% RSLogix 500 project ML02B JOB 10 NL.RSS, saved by version 10.00.00.00 %
PROJECT "UNTITLED"    % processor: Bul.1763 MicroLogix 1100 Series B %

PROGRAM FILES
  LAD 2   5 rungs

DATA FILES
  O0 OUTPUT  4 elements
  I1 INPUT  6 elements
  S2 STATUS  66 elements
  B3 BINARY  1 elements
  T4 TIMER  1 elements
  C5 COUNTER  1 elements
  R6 CONTROL  1 elements
  N7 INTEGER  1 elements
  F8 FLOAT  1 elements

LADDER 2
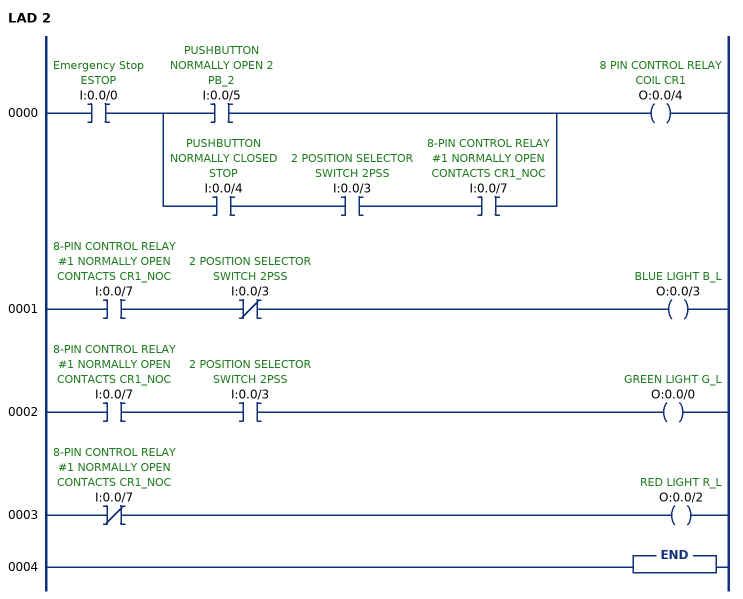
% Rung: 0 %
SOR XIC I:0.0/0 BST XIC I:0.0/5 NXB XIC I:0.0/4 XIC I:0.0/3 XIC I:0.0/7 BND OTE O:0.0/4 EOR
%   I:0.0/0  ESTOP  "Emergency Stop" %
%   I:0.0/5  PB_2  "PUSHBUTTON NORMALLY OPEN 2" %
%   I:0.0/4  STOP  "PUSHBUTTON NORMALLY CLOSED" %
%   I:0.0/3  2PSS  "2 POSITION SELECTOR SWITCH" %
%   I:0.0/7  CR1_NOC  "8-PIN CONTROL RELAY #1 NORMALLY OPEN CONTACTS" %
%   O:0.0/4  CR1  "8 PIN CONTROL RELAY COIL" %
% Rung: 1 %
SOR XIC I:0.0/7 XIO I:0.0/3 OTE O:0.0/3 EOR
%   I:0.0/7  CR1_NOC  "8-PIN CONTROL RELAY #1 NORMALLY OPEN CONTACTS" %
%   I:0.0/3  2PSS  "2 POSITION SELECTOR SWITCH" %
%   O:0.0/3  B_L  "BLUE LIGHT" %
% Rung: 2 %
SOR XIC I:0.0/7 XIC I:0.0/3 OTE O:0.0/0 EOR
%   I:0.0/7  CR1_NOC  "8-PIN CONTROL RELAY #1 NORMALLY OPEN CONTACTS" %
%   I:0.0/3  2PSS  "2 POSITION SELECTOR SWITCH" %
%   O:0.0/0  G_L  "GREEN LIGHT" %
% Rung: 3 %
SOR XIO I:0.0/7 OTE O:0.0/2 EOR
%   I:0.0/7  CR1_NOC  "8-PIN CONTROL RELAY #1 NORMALLY OPEN CONTACTS" %
%   O:0.0/2  R_L  "RED LIGHT" %
% Rung: 4 %
SOR END EOR

OTHER DOCUMENTED ADDRESSES
  I:0.0/1  3PSS_A  "3 Position Selector Switch, Posiition A"
  I:0.0/2  3PSS_B  "3 POSITION SELECTOR SWITCH, POSITION B"
  I:0.0/6  PB_3  "PUSHBUTTON NORMALLY OPEN 3"
  I:0.0/8  CR2_NOC  "11-PIN RELAY NORMALLY OPEN CONTACTS"
  I:0.0/9  MS_1  "3 PHASE MOTOR STARTER. CONTACTS & OVERLOAD"
  O:0.0/1  Y_L  "YELLOW LIGHT"
  O:0.0/5  CR2  "11 PIN RELAY COIL"
